FUNCTION BytesToUint : UINT
VAR_INPUT
	b1	: BYTE;
	b2	: BYTE;
END_VAR

BytesToUint := TO_UINT(b2) 
			+ TO_UINT(b1) * 256;

END_FUNCTION

(* stored: Version 1.1.0.1
   POU BytesToUint: Id {9bf4e454-9ed4-49a3-bd75-928b49e5b1ac}, SpecialFunc None *)
